Fanuc KAREL source: kt00611.KL

-- PROVISIONAL review KL for V940-1; original PC SHA256 ce2ceeba68ece7eee7e626faadf1c460237189e9abb7a2aebedcf35f5e3eba2f
-- Incomplete behavior may be omitted. Consult companion uncertainty JSON. Do not deploy.
PROGRAM KT00611
%NOLOCKGROUP
VAR
  R1 : REAL
  R2 : REAL
  OUT : REAL
BEGIN
  -- V9_ZERO_TABLE_METADATA_HINT layout=0001; no indexed target words; source/name/runtime held
  -- UNRESOLVED_PC offsets 5-16; opcodes 2E,23
  -- UNRESOLVED_PC offsets 21-32; opcodes 2E,23
  -- UNRESOLVED_PC offsets 37-48; opcodes 2E,23
  -- UNRESOLVED_PC offsets 53-64; opcodes 2E,23
  -- UNRESOLVED_PC offsets 69-81; opcodes 21,23
  -- UNRESOLVED_PC offsets 86-90; opcodes 7F
END KT00611
